FUNCTION_BLOCK TT_TEST (* Basic Function Block Type *)
  (* Standard: 61499-2 *)
  (* Version 0.3, 2009-09-15, JHC, Holobloc Inc, Changed transition priorities. *)
  (* Version 0.2, 2003-12-04, JHC, Rockwell Automation, Renamed for better indexing. *)
  (* Version 0.1, 2002-11-05, JHC, Rockwell Automation, Corrected missing ST element in Algorithm REQ. *)
  (* Version 0.0, 2000-05-30, JHC, Rockwell Automation *)
  PACKAGE fb.rt.template;
  IMPORT fb.datatype.*;
  IMPORT fb.rt.*;
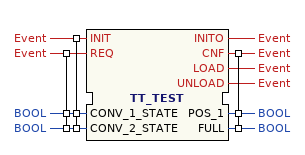
  EVENT_INPUT
    INIT WITH CONV_1_STATE, CONV_2_STATE; (* Initialization Request *)
    REQ WITH CONV_1_STATE, CONV_2_STATE; (* Normal Execution Request *)
  END_EVENT
  EVENT_OUTPUT
    INITO; (* Initialization Confirm *)
    CNF WITH POS_1, FULL;
    LOAD;
    UNLOAD;
  END_EVENT
  VAR_INPUT
    CONV_1_STATE : BOOL;
    CONV_2_STATE : BOOL;
  END_VAR
  VAR_OUTPUT
    POS_1 : BOOL;
    FULL : BOOL;
  END_VAR
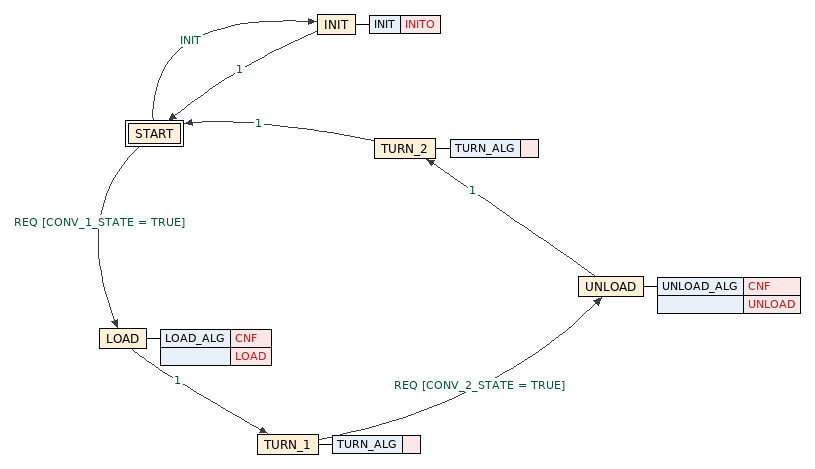
  EC_STATES
    START; (* Initial State *)
    INIT : INIT -> INITO; (* Initialization *)
    LOAD : LOAD_ALG -> CNF, -> LOAD;
    TURN_1 : TURN_ALG;
    UNLOAD : UNLOAD_ALG -> CNF, -> UNLOAD;
    TURN_2 : TURN_ALG;
  END_STATES
  EC_TRANSITIONS
    START TO INIT := INIT;
    INIT TO START := 1;
    START TO LOAD := REQ [CONV_1_STATE = TRUE];
    LOAD TO TURN_1 := 1;
    TURN_1 TO UNLOAD := REQ [CONV_2_STATE = TRUE];
    UNLOAD TO TURN_2 := 1;
    TURN_2 TO START := 1;
  END_TRANSITIONS
  ALGORITHM INIT IN ST: (* Initialization algorithm *)
POS_1 := TRUE;
FULL := FALSE;
  END_ALGORITHM
  ALGORITHM LOAD_ALG IN ST:
FULL := TRUE;
  END_ALGORITHM
  ALGORITHM TURN_ALG IN ST:
POS_1 := NOT POS_1;
  END_ALGORITHM
  ALGORITHM UNLOAD_ALG IN ST:
FULL := FALSE;
  END_ALGORITHM
END_FUNCTION_BLOCK
